FUNCTION_BLOCK FB_Shelly_Pro4PM
VAR_INPUT
	bStart				: BOOL;
	tDelayRequest		: TIME := T#3S;	//Timer for delay before start with the next read or write Request
	sHostname			: STRING(255);		//Hostname or IP Adress from the Server
END_VAR

VAR_IN_OUT
END_VAR

VAR_OUTPUT
	bValidResult				: BOOL;															//Valid Result received from Server
    bBusy						: BOOL;															//Function is Busy
    bError						: BOOL;															//Error sucess
	bDone						: BOOL;															//True after the decoding from the received Json File
	bConnected					: BOOL;															//Connection to the Server
	lrpowerP1					: LREAL;														//Received Value
	lrvoltageP1					: LREAL;														//Received Value
	lrenergyP1					: LREAL;														//Received Value
	lrpowerP2					: LREAL;														//Received Value
	lrvoltageP2					: LREAL;														//Received Value
	lrenergyP2					: LREAL;
	lrpowerP3					: LREAL;														//Received Value
	lrvoltageP3					: LREAL;														//Received Value
	lrenergyP3					: LREAL;
	lrpowerP4					: LREAL;														//Received Value
	lrvoltageP4					: LREAL;														//Received Value
	lrenergyP4					: LREAL;	
	hrErrorCode       			: HRESULT;														//Error Result from Http Client
END_VAR

VAR
	fbClient					: FB_IotHttpClient;
	fbHttpGet					: FB_Shelly_Pro4PM_Helper;
	timStartRequest				: TON;															//Timer to Start the Request
	FPStartRequest				: R_TRIG;														//Internal positive Edge
	FPDone						: R_TRIG;														//Internal positive Edge
	FNStart						: F_TRIG;														//Internal negative Edge
END_VAR

(*------------------------------------------------------------------------------------Configure HTTP Client------------------------------------------------------------------------------------------------------*)

fbClient.sHostName := sHostname;
fbClient.tConnectionTimeout := tDelayRequest;

IF NOT fbClient.bConfigured THEN 
	fbClient.nHostPort:= 80;
	fbClient.bKeepAlive := TRUE;
	fbClient.tConnectionTimeout := T#2S;
END_IF


//Timer to start the Request
FPStartRequest(CLK:= bStart, Q=> );
	timStartRequest(IN:= fbClient.bConfigured AND bStart AND NOT timStartRequest.Q, PT:= tDelayRequest, Q=> , ET=> );
		IF ((timStartRequest.Q AND NOT bBusy) OR (FPStartRequest.Q AND NOT bBusy AND fbClient.bConfigured)) THEN fbHttpGet.bSend := TRUE; END_IF

				
//Http Get Function
fbHttpGet(
	lrapowerP1 => lrpowerP1, 
	lrvoltageP1 => lrvoltageP1, 
	lraenergyP1 => lrenergyP1,
	lrapowerP2 => lrpowerP2, 
	lrvoltageP2 => lrvoltageP2, 
	lraenergyP2 => lrenergyP2,
	lrapowerP3 => lrpowerP3, 
	lrvoltageP3 => lrvoltageP3, 
	lraenergyP3 => lrenergyP3,
	lrapowerP4 => lrpowerP4, 
	lrvoltageP4 => lrvoltageP4, 
	lraenergyP4 => lrenergyP4, 
	bSend:= , 
	fbClient:= fbClient, 
	bBusy=> bBusy, 
	bError=> ,
	sContentS0=> ,
	sContentS1=> ,
	sContentS2=> ,
	sContentS3=> );


fbHttpGet.bSend := FALSE;

FPDone(CLK:= bDone, Q=> );

(*
//Http Client
FNStart(CLK:= bStart, Q=> );
	IF FNStart.Q THEN fbClient.Disconnect(); END_IF
*)

fbClient.Execute();

//Error
IF fbHttpGet.bError OR fbClient.bError THEN bError := TRUE; ELSE bError := FALSE; END_IF	
	hrErrorCode := fbClient.hrErrorCode;

END_FUNCTION_BLOCK

(* stored: Version 1.1.0.1, ProductVersion 3.1.4024.9
   POU FB_Shelly_Pro4PM: Id {4fb64124-ca1a-4f6d-b795-35461972a121}, SpecialFunc None *)
